// TIA Portal V17 export
// export: Created 2022-07-20T07:02:36.3395735Z, ExportSetting WithDefaults, DisplayName Totally Integrated Automation Portal, DisplayVersion V17, DisplayName TIA Portal Openness, DisplayVersion V17, DisplayName TIA Portal Version Control Interface, DisplayVersion V17, DisplayName SINAMICS Startdrive Advanced, DisplayVersion V17, DisplayName SINAMICS Startdrive G130, G150, S120, S150, SINAMICS MV, S210, DisplayVersion V17, DisplayName SINAMICS Startdrive G110M, G120, G120C, G120D, G120P, G115D, DisplayVersion V17, DisplayName STEP 7 Professional, DisplayVersion V17, DisplayName STEP 7 Safety, DisplayVersion V17, DisplayName WinCC Advanced, DisplayVersion V17
VAR_GLOBAL   // PLC tag table "OMAC_STATE"
END_VAR
VAR_GLOBAL CONSTANT   // user constants
   OMAC_STATE_ABORTED : USInt := 1;
   OMAC_STATE_CLEARING : USInt := 2;
   OMAC_STATE_STOPPED : USInt := 3;
   OMAC_STATE_RESETTING : USInt := 4;
   OMAC_STATE_IDLE : USInt := 5;
   OMAC_STATE_STARTING : USInt := 6;
   OMAC_STATE_EXECUTE : USInt := 7;
   OMAC_STATE_HOLDING : USInt := 8;
   OMAC_STATE_HELD : USInt := 9;
   OMAC_STATE_UNHOLDING : USInt := 10;
   OMAC_STATE_SUSPENDING : USInt := 11;
   OMAC_STATE_SUSPENDED : USInt := 12;
   OMAC_STATE_UNSUSPENDING : USInt := 13;
   OMAC_STATE_COMPLETING : USInt := 14;
   OMAC_STATE_COMPLETE : USInt := 15;
   OMAC_STATE_STOPPING : USInt := 16;
   OMAC_STATE_ABORTING : USInt := 17;
END_VAR
